FUNCTION_BLOCK FB_DynamicWeighing
VAR_INPUT
	aInput : ARRAY[1..cOversamples] OF LREAL;
	//aInput : LREAL;
END_VAR
VAR_OUTPUT
	bError : BOOL;
	ipResultMessage : I_TcMessage;
	bNewResult : BOOL;	
	bValidMeasurement : BOOL;	
	fWeight : LREAL;
	fLastWeight : LREAL;
	fStd : LREAL;
	fLastStd : LREAL;
END_VAR
VAR
// Filter
	stParamsComboFilter : ST_WG_ComboFilter := 
	(
		nOrder:= GVL_WEIGHING_IHM.nFilterOrder,
		fCutoff:=GVL_WEIGHING_IHM.rCutOff,
		fSamplingRate:=TO_LREAL(GVL_WEIGHING_IHM.cSamplingRate),
		nSamplesToFilter:=GVL_WEIGHING_IHM.nSamplesToFilter,
		bReset := GVL_WEIGHING_IHM.bResetFilter
	);
	
	fbComboFilter : FB_WG_ComboFilter:=(stConfig := stParamsComboFilter);

// Scaling
	stParamsScale : ST_WG_Scaling :=
	(	
		fRawLow:=GVL_WEIGHING_IHM.fRawLow,
		fReferenceLow:=GVL_WEIGHING_IHM.fReferenceLow,
		fRawHigh:=GVL_WEIGHING_IHM.fRawHigh,
		fReferenceHigh:=GVL_WEIGHING_IHM.fReferenceHigh
	);	
	
	nNumCalibrationSamples : UDINT := 100;
	nNumTareSamples : UDINT := 100;
	fbScale : FB_WG_Scaling:=(stConfig:=stParamsScale, eTraceLevel:=TcEventSeverity.Info);
	
// Weighing
	stParamsWeighing : ST_WG_Weighing := 
	(
		nWindowLength:=GVL_WEIGHING_IHM.nWindowLenght,
		Validation:=(nValidationSamples:=GVL_WEIGHING_IHM.nValidationSamplesValidation,
					  fThresholdWeight:=GVL_WEIGHING_IHM.fThresholdWeightValidation, 
					  fMaxStd:=GVL_WEIGHING_IHM.fMaxStdValidation,
					  fMaxWeightDeviation:=GVL_WEIGHING_IHM.fMaxWeightDeviationValidation),
					  
		AutoTare:=(nValidationSamples:=GVL_WEIGHING_IHM.nValidationSamplesAutoTare,
				    fThresholdWeight:=GVL_WEIGHING_IHM.fThresholdWeightAutoTare,
					fMaxStd:=GVL_WEIGHING_IHM.fMaxStdAutoTare,
					fMaxWeightDeviation:=GVL_WEIGHING_IHM.fMaxWeightDeviationAutoTare)
	);
	
	fbWeighing : FB_WG_Weighing:=(stConfig:=stParamsWeighing);
	
// Helper
	aOutFilter : ARRAY[1..cOversamples] OF LREAL; // Stage1 PTn filter, Stage2 MovAvg Filter
	aOutScaling : ARRAY[1..cOversamples] OF LREAL; // Scaling
	reconfigureFilter : R_TRIG;
	reconfigureWeighing : R_TRIG;
	calibrateReferenceLow : R_TRIG;
	calibrateReferenceHigh : R_TRIG;
	applyCalibration : R_TRIG;
	tare : R_TRIG;
	
// Control
	// Reconfigure
	bReconfigureFilter : BOOL := FALSE;
	bReconfigureWeighing : BOOL := FALSE;
	// Calibration
	fCalibrateReferenceLow : LREAL := 417;
	fCalibrateReferenceHigh : LREAL := 1215;
	bCalibrateReferenceLow : BOOL := FALSE;		// e.g. ref: 417	| raw: 175000
	bCalibrateReferenceHigh : BOOL := FALSE;	// e.g. ref: 1215	| raw: 525000	
	bApplyCalibration : BOOL := FALSE;
	bAcceptCalibration : BOOL := TRUE;
	// Tare
	bTare : BOOL := FALSE;
	fMaxTotalTareLimit : LREAL := 40.0; // set error if total taring amount exceeds the limit
	eAutoTareType : E_WG_AutoTareType := E_WG_AutoTareType.eContinously;
	
	
	//UserMessage
	fbCustomMessage : FB_TcMessage;
END_VAR

(* IHM params *)
stParamsScale.fRawLow 			:= GVL_WEIGHING_IHM.fRawLow;
stParamsScale.fReferenceLow 	:= GVL_WEIGHING_IHM.fReferenceLow;
stParamsScale.fRawHigh		 	:= GVL_WEIGHING_IHM.fRawHigh;
stParamsScale.fReferenceHigh	:= GVL_WEIGHING_IHM.fReferenceHigh;



nNumCalibrationSamples 	:= GVL_WEIGHING_IHM.nNumCalibrationSamples;
nNumTareSamples 		:= GVL_WEIGHING_IHM.nNumTareSamples;
fCalibrateReferenceLow 	:= GVL_WEIGHING_IHM.fCalibrateReferenceLow;
fCalibrateReferenceHigh := GVL_WEIGHING_IHM.fCalibrateReferenceHigh;
bAcceptCalibration		:= GVL_WEIGHING_IHM.bAcceptCalibration;
bTare					:= GVL_WEIGHING_IHM.bTare;
fMaxTotalTareLimit		:= GVL_WEIGHING_IHM.fMaxTotalTareLimit;
eAutoTareType			:= GVL_WEIGHING_IHM.eAutoTareType;

bError := FALSE;
CommandTrigger();

// Reconfigure
IF reconfigureFilter.Q AND_THEN NOT fbComboFilter.Configure(stParamsComboFilter) THEN
	SetError(fbComboFilter);
END_IF

stParamsWeighing.nWindowLength := GVL_WEIGHING_IHM.nWindowLenght;
stParamsWeighing.Validation.fMaxStd := GVL_WEIGHING_IHM.fMaxStdValidation;
stParamsWeighing.Validation.fMaxWeightDeviation := GVL_WEIGHING_IHM.fMaxWeightDeviationValidation;
stParamsWeighing.Validation.fRelativeWeightLimit := GVL_WEIGHING_IHM.fRelativeWeightLimit;
stParamsWeighing.Validation.fThresholdWeight := GVL_WEIGHING_IHM.fThresholdWeightValidation;
stParamsWeighing.Validation.nValidationSamples := GVL_WEIGHING_IHM.nValidationSamplesValidation;

IF reconfigureWeighing.Q AND_THEN NOT fbWeighing.Configure(stParamsWeighing) THEN
	SetError(fbWeighing);
END_IF

// Calibration	 
IF calibrateReferenceLow.Q AND_THEN NOT fbScale.CalibrateRefLow(nNumCalibrationSamples, fCalibrateReferenceLow) THEN
	SetError(fbScale);
END_IF

IF calibrateReferenceHigh.Q AND_THEN NOT fbScale.CalibrateRefHigh(nNumCalibrationSamples, fCalibrateReferenceHigh) THEN
	SetError(fbScale);
END_IF

IF applyCalibration.Q AND_THEN NOT fbScale.ApplyCalibration(bAcceptCalibration) THEN
	SetError(fbScale);
END_IF

// Tare
IF tare.Q AND_THEN NOT fbScale.Tare(nNumTareSamples) THEN
	SetError(fbScale);
END_IF

// Perform taring process continously if fbWeighing.fAutoTareOffset is not zero
// Careful: ST_WG_Weighing_AutoTare.nValidationSamples should be large enough, to find the best tare weight.
// Execute AutoTare
IF NOT fbWeighing.AutoTare(fbScale, eAutoTareType)THEN
	SetError(fbWeighing);
END_IF

IF ABS(fbScale.fCurrentTareOffset - fbWeighing.fAutoTareOffset) > fMaxTotalTareLimit THEN
	SetCustomWarning(fbCustomMessage, 'Total taring amount exceeds the limit. Please check the weighing machine!');
END_IF


// Execute weighing
IF NOT fbComboFilter.Call(ADR(aInput), SIZEOF(aInput), ADR(aOutFilter), SIZEOF(aOutFilter)) THEN
	SetError(fbComboFilter);
END_IF

IF NOT fbScale.Call(ADR(aOutFilter), SIZEOF(aOutFilter), ADR(aOutScaling), SIZEOF(aOutScaling)) THEN
	SetError(fbScale);
END_IF

IF NOT fbWeighing.Call(ADR(aOutScaling), SIZEOF(aOutScaling)) THEN
	SetError(fbWeighing);
END_IF

// Assign results
AssignResults();

METHOD AssignResults : BOOL
VAR_INPUT
END_VAR
bNewResult := fbWeighing.bNewResult;	
bValidMeasurement := fbWeighing.bValidMeasurement;	
fWeight := fbWeighing.fWeight;
fLastWeight := fbWeighing.fLastWeight;
fStd := fbWeighing.fStd;
fLastStd := fbWeighing.fLastStd;
END_METHOD

METHOD CommandTrigger : BOOL
VAR_INPUT
END_VAR
reconfigureFilter(CLK:=bReconfigureFilter OR GVL_WEIGHING_IHM.bReconfigureFilter);
reconfigureWeighing(CLK:=bReconfigureWeighing OR GVL_WEIGHING_IHM.bReconfigureWeighing);
calibrateReferenceLow(CLK:=bCalibrateReferenceLow OR GVL_WEIGHING_IHM.bCalibrateReferenceLow);
calibrateReferenceHigh(CLK:=bCalibrateReferenceHigh OR GVL_WEIGHING_IHM.bCalibrateReferenceHigh);
applyCalibration(CLK:=bApplyCalibration OR GVL_WEIGHING_IHM.bApplyCalibration);
tare(CLK:=bTare);
END_METHOD

METHOD SetCustomWarning : BOOL
VAR_INPUT
	fb : REFERENCE TO FB_TcMessage;
	sText : STRING;
END_VAR
VAR
END_VAR
THIS^.bError := TRUE;
fb.CreateEx(TC_EVENTS.TcWeighingEventClass.Warning_InvalidThreshold,0);
fb.ipArguments.Clear();
fb.ipArguments.AddString(sText);
fb.Send(0);
THIS^.ipResultMessage := fb;
END_METHOD

METHOD SetError : BOOL
VAR_INPUT
	fb : REFERENCE TO _FB_WG_BasicImplementationAlgorithm;
END_VAR
THIS^.bError := fb.bError;
THIS^.ipResultMessage := fb.ipResultMessage;
END_METHOD

END_FUNCTION_BLOCK

(* stored: Version 1.1.0.1, ProductVersion 3.1.4026.17
   POU FB_DynamicWeighing: Id {e36022e2-584d-45fe-972e-e8dc27e347b5}, SpecialFunc None
   Method AssignResults: Id {5338b36c-b8c1-43fa-b63f-6f36aa7572dc}
   Method CommandTrigger: Id {9433b606-638b-4587-9c83-7d2d5401227f}
   Method SetCustomWarning: Id {a2106cc0-f7c6-4d66-842d-6668ef5cb125}
   Method SetError: Id {505b0742-9aaf-4cd9-b34c-4a783691ae12} *)
